Fanuc KAREL source: kt00158.compact.KL

PROGRAM KT00158
%STACKSIZE=65535
%PRIORITY=65535
%NOLOCKGROUP
VAR
H1 : ARRAY[2] OF SHORT
Y2 : ARRAY[2] OF BYTE
OUT : REAL
BEGIN
H1[1]=2
Y2[1]=3
OUT=((H1[1] DIV Y2[1]))
END KT00158
